{attribute addProperty BoxType "EP4378-1022-0017"}
{attribute addProperty Id "DI_X01_Pin4_InputAT %I*DI_X01_Pin4_Input_E4AEF59E810DI_X02_Pin4_InputAT %I*DI_X02_Pin4_Input_E4AEF59E810DI_X03_Pin4_InputAT %I*DI_X03_Pin4_Input_E4AEF59E810DI_X04_Pin4_InputAT %I*DI_X04_Pin4_Input_E4AEF59E810DI_X05_Pin4_InputAT %I*DI_X05_Pin4_Input_E4AEF59E810DI_X06_Pin4_InputAT %I*DI_X06_Pin4_Input_E4AEF59E810DI_X07_Pin4_InputAT %I*DI_X07_Pin4_Input_E4AEF59E810DI_X08_Pin4_InputAT %I*DI_X08_Pin4_Input_E4AEF59E810AI_X01_Pin2_StandardAT %I*AI_X01_Pin2_Standard_087F71C73240AI_X02_Pin2_StandardAT %I*AI_X02_Pin2_Standard_087F71C73240AI_X05_Pin2_StandardAT %I*AI_X05_Pin2_Standard_087F71C73240AI_X06_Pin2_StandardAT %I*AI_X06_Pin2_Standard_087F71C73240DO_X01_Pin4_OutputAT %Q*DO_X01_Pin4_Output_7F374EB0810DO_X02_Pin4_OutputAT %Q*DO_X02_Pin4_Output_7F374EB0810DO_X03_Pin4_OutputAT %Q*DO_X03_Pin4_Output_7F374EB0810DO_X04_Pin4_OutputAT %Q*DO_X04_Pin4_Output_7F374EB0810DO_X05_Pin4_OutputAT %Q*DO_X05_Pin4_Output_7F374EB0810DO_X06_Pin4_OutputAT %Q*DO_X06_Pin4_Output_7F374EB0810DO_X07_Pin4_OutputAT %Q*DO_X07_Pin4_Output_7F374EB0810DO_X08_Pin4_OutputAT %Q*DO_X08_Pin4_Output_7F374EB0810AO_X01_Pin5_StandardAT %Q*AO_X01_Pin5_Standard_F57FA4F91620AO_X02_Pin5_StandardAT %Q*AO_X02_Pin5_Standard_F57FA4F91620AO_X05_Pin5_StandardAT %Q*AO_X05_Pin5_Standard_F57FA4F91620AO_X06_Pin5_StandardAT %Q*AO_X06_Pin5_Standard_F57FA4F91620WcStateAT %I*WcState_98A4DF7520.250InfoDataAT %I*InfoData_BC63D37F80100"}
{attribute addProperty CRC "2302991572"}
{attribute addProperty SizeInBites "402"}
{attribute addProperty SizeInBytes "50.25"}
TYPE EP4378_B0B1C4E6 :
STRUCT
	{attribute addProperty Name "DI_X01_Pin4_Input"}
	DI_X01_Pin4_Input : DI_X01_Pin4_Input_E4AEF59E;
	{attribute addProperty Name "DI_X02_Pin4_Input"}
	DI_X02_Pin4_Input : DI_X02_Pin4_Input_E4AEF59E;
	{attribute addProperty Name "DI_X03_Pin4_Input"}
	DI_X03_Pin4_Input : DI_X03_Pin4_Input_E4AEF59E;
	{attribute addProperty Name "DI_X04_Pin4_Input"}
	DI_X04_Pin4_Input : DI_X04_Pin4_Input_E4AEF59E;
	{attribute addProperty Name "DI_X05_Pin4_Input"}
	DI_X05_Pin4_Input : DI_X05_Pin4_Input_E4AEF59E;
	{attribute addProperty Name "DI_X06_Pin4_Input"}
	DI_X06_Pin4_Input : DI_X06_Pin4_Input_E4AEF59E;
	{attribute addProperty Name "DI_X07_Pin4_Input"}
	DI_X07_Pin4_Input : DI_X07_Pin4_Input_E4AEF59E;
	{attribute addProperty Name "DI_X08_Pin4_Input"}
	DI_X08_Pin4_Input : DI_X08_Pin4_Input_E4AEF59E;
	{attribute addProperty Name "AI_X01_Pin2_Standard"}
	AI_X01_Pin2_Standard : AI_X01_Pin2_Standard_087F71C7;
	{attribute addProperty Name "AI_X02_Pin2_Standard"}
	AI_X02_Pin2_Standard : AI_X02_Pin2_Standard_087F71C7;
	{attribute addProperty Name "AI_X05_Pin2_Standard"}
	AI_X05_Pin2_Standard : AI_X05_Pin2_Standard_087F71C7;
	{attribute addProperty Name "AI_X06_Pin2_Standard"}
	AI_X06_Pin2_Standard : AI_X06_Pin2_Standard_087F71C7;
	{attribute addProperty Name "DO_X01_Pin4_Output"}
	DO_X01_Pin4_Output : DO_X01_Pin4_Output_7F374EB0;
	{attribute addProperty Name "DO_X02_Pin4_Output"}
	DO_X02_Pin4_Output : DO_X02_Pin4_Output_7F374EB0;
	{attribute addProperty Name "DO_X03_Pin4_Output"}
	DO_X03_Pin4_Output : DO_X03_Pin4_Output_7F374EB0;
	{attribute addProperty Name "DO_X04_Pin4_Output"}
	DO_X04_Pin4_Output : DO_X04_Pin4_Output_7F374EB0;
	{attribute addProperty Name "DO_X05_Pin4_Output"}
	DO_X05_Pin4_Output : DO_X05_Pin4_Output_7F374EB0;
	{attribute addProperty Name "DO_X06_Pin4_Output"}
	DO_X06_Pin4_Output : DO_X06_Pin4_Output_7F374EB0;
	{attribute addProperty Name "DO_X07_Pin4_Output"}
	DO_X07_Pin4_Output : DO_X07_Pin4_Output_7F374EB0;
	{attribute addProperty Name "DO_X08_Pin4_Output"}
	DO_X08_Pin4_Output : DO_X08_Pin4_Output_7F374EB0;
	{attribute addProperty Name "AO_X01_Pin5_Standard"}
	AO_X01_Pin5_Standard : AO_X01_Pin5_Standard_F57FA4F9;
	{attribute addProperty Name "AO_X02_Pin5_Standard"}
	AO_X02_Pin5_Standard : AO_X02_Pin5_Standard_F57FA4F9;
	{attribute addProperty Name "AO_X05_Pin5_Standard"}
	AO_X05_Pin5_Standard : AO_X05_Pin5_Standard_F57FA4F9;
	{attribute addProperty Name "AO_X06_Pin5_Standard"}
	AO_X06_Pin5_Standard : AO_X06_Pin5_Standard_F57FA4F9;
	{attribute addProperty Name "WcState"}
	WcState : WcState_98A4DF75;
	{attribute addProperty Name "InfoData"}
	InfoData : InfoData_BC63D37F;
END_STRUCT
END_TYPE

(* stored: Version 1.2.0.0, ProductVersion 3.1.4024.9
   DUT EP4378_B0B1C4E6: Id {851edf02-2a65-4775-ba4b-2799f57902b7} *)
